(* IEC 61131-3 sources: RL_MAR/experiments/comparison/llm4plc/results/gpt-4o_20260507_114630/20260507_122226, 4 files *)

(* ---- generated_code_iteration_0.st ---- *)
plaintext
START_ST
FUNCTION_BLOCK AGVControlSystem
VAR_INPUT
    MaterialRequest : INT; (* New material handling request *)
END_VAR
VAR_OUTPUT
    AGV1_Ready : BOOL := TRUE; (* AGV 1 ready status *)
    AGV2_Ready : BOOL := TRUE; (* AGV 2 ready status *)
    AGV3_Ready : BOOL := TRUE; (* AGV 3 ready status *)
END_VAR
VAR
    state : INT := 0; (* Current state *)
    prevState : INT := 0; (* Previous state *)
    MaterialQueue : ARRAY[1..10] OF INT; (* FIFO queue for material requests *)
    queueHead : INT := 1; (* Points to the first element in the queue *)
    queueTail : INT := 0; (* Points to the last element in the queue *)
    AGVPosition : ARRAY[1..3] OF INT := [0, 0, 0]; (* Real-time AGV positions *)
    AGVStatus : ARRAY[1..3] OF BOOL := [TRUE, TRUE, TRUE]; (* Operational status of AGVs *)
    currentTask : ARRAY[1..3] OF INT := [0, 0, 0]; (* Task currently assigned to each AGV *)
    errorFlag : BOOL := FALSE; (* Error detection flag *)
    i : INT; (* Loop counter *)
END_VAR

(* Function to add a new material request to the queue *)
FUNCTION AddToQueue : BOOL
VAR_INPUT
    MaterialRequest : INT; (* Material request to be added *)
END_VAR
VAR
    success : BOOL := FALSE; (* Indicates if the operation was successful *)
END_VAR
IF queueTail < 10 THEN
    queueTail := queueTail + 1;
    MaterialQueue[queueTail] := MaterialRequest;
    success := TRUE;
ELSE
    success := FALSE; (* Queue overflow detected *)
END_IF
RETURN success;
END_FUNCTION

(* Function to assign tasks to AGVs based on priority and readiness *)
FUNCTION AssignTask : BOOL
VAR
    success : BOOL := FALSE; (* Indicates if the operation was successful *)
END_VAR
FOR i := 1 TO 3 DO
    IF AGVStatus[i] = TRUE AND queueHead <= queueTail THEN
        currentTask[i] := MaterialQueue[queueHead];
        AGVStatus[i] := FALSE; (* AGV is now working *)
        queueHead := queueHead + 1;
        success := TRUE;
        EXIT; (* Assign task to the highest priority AGV and exit *)
    END_IF
END_FOR
RETURN success;
END_FUNCTION

(* Function to update AGV position based on task progress *)
FUNCTION UpdateAGVPosition : BOOL
VAR_INPUT
    AGVIndex : INT; (* Index of the AGV to update *)
END_VAR
VAR
    success : BOOL := FALSE; (* Indicates if the operation was successful *)
END_VAR
IF AGVIndex >= 1 AND AGVIndex <= 3 THEN
    AGVPosition[AGVIndex] := AGVPosition[AGVIndex] + 1; (* Simulate position update *)
    IF AGVPosition[AGVIndex] < 0 THEN
        errorFlag := TRUE; (* Invalid position detected *)
        success := FALSE;
    ELSE
        success := TRUE;
    END_IF
END_IF
RETURN success;
END_FUNCTION

(* Function to reset AGV status after task completion *)
FUNCTION ResetAGVStatus : BOOL
VAR_INPUT
    AGVIndex : INT; (* Index of the AGV to reset *)
END_VAR
VAR
    success : BOOL := FALSE; (* Indicates if the operation was successful *)
END_VAR
IF AGVIndex >= 1 AND AGVIndex <= 3 THEN
    AGVStatus[AGVIndex] := TRUE; (* Reset AGV status to ready *)
    currentTask[AGVIndex] := 0; (* Clear the current task *)
    AGVPosition[AGVIndex] := 0; (* Reset position *)
    success := TRUE;
END_IF
RETURN success;
END_FUNCTION

(* Function to handle errors *)
FUNCTION HandleError : BOOL
VAR
    success : BOOL := FALSE; (* Indicates if the operation was successful *)
END_VAR
IF queueTail > 10 THEN
    queueTail := 10; (* Correct queue overflow *)
    errorFlag := TRUE;
    success := TRUE;
ELSIF errorFlag THEN
    errorFlag := FALSE; (* Clear error flag *)
    success := TRUE;
END_IF
RETURN success;
END_FUNCTION

(* Main logic for state transitions *)
CASE state OF
    0: (* IDLE *)
        IF MaterialRequest > 0 AND queueTail < 10 THEN
            prevState := state;
            state := 1; (* Transition to ADD_REQUEST_TO_QUEUE *)
        END_IF;
    1: (* ADD_REQUEST_TO_QUEUE *)
        IF AddToQueue(MaterialRequest) THEN
            prevState := state;
            state := 2; (* Transition to ASSIGN_TASK_TO_AGV *)
        ELSE
            prevState := state;
            state := 5; (* Transition to ERROR_HANDLING *)
        END_IF;
    2: (* ASSIGN_TASK_TO_AGV *)
        IF AssignTask() THEN
            prevState := state;
            state := 3; (* Transition to AGV_WORKING *)
        END_IF;
    3: (* AGV_WORKING *)
        FOR i := 1 TO 3 DO
            IF NOT AGVStatus[i] THEN
                IF UpdateAGVPosition(i) THEN
                    (* Check if task is completed *)
                    IF AGVPosition[i] >= 10 THEN
                        prevState := state;
                        state := 4; (* Transition to RESET_AGV_STATUS *)
                    END_IF;
                ELSE
                    prevState := state;
                    state := 5; (* Transition to ERROR_HANDLING *)
                END_IF;
            END_IF;
        END_FOR;
    4: (* RESET_AGV_STATUS *)
        FOR i := 1 TO 3 DO
            IF NOT AGVStatus[i] THEN
                IF ResetAGVStatus(i) THEN
                    prevState := state;
                    state := 0; (* Transition to IDLE *)
                END_IF;
            END_IF;
        END_FOR;
    5: (* ERROR_HANDLING *)
        IF HandleError() THEN
            prevState := state;
            state := 0; (* Transition to IDLE *)
        END_IF;
END_CASE;
END_FUNCTION_BLOCK
END_ST

(* ---- generated_code_iteration_1.st ---- *)
START_REASON
The feedback indicates that the `AddToQueue` function declaration is incorrect. Specifically, the function's output variable is improperly defined as `AddToQueue: BOOL;`. In Structured Text (ST), functions must use `VAR_OUTPUT` to declare output variables, not directly in the function header. This syntax error caused the CODESYS compiler validation to fail.

To resolve this issue, I will modify the function declaration to properly define the output variable using `VAR_OUTPUT`. Additionally, I will review the code for similar issues in other functions and ensure compliance with ST syntax standards.
END_REASON

START_ST
FUNCTION_BLOCK AGVControlSystem
VAR_INPUT
    MaterialRequest : INT; (* New material handling request *)
END_VAR
VAR_OUTPUT
    AGV1_Ready : BOOL := TRUE; (* AGV 1 ready status *)
    AGV2_Ready : BOOL := TRUE; (* AGV 2 ready status *)
    AGV3_Ready : BOOL := TRUE; (* AGV 3 ready status *)
END_VAR
VAR
    state : INT := 0; (* Current state *)
    prevState : INT := 0; (* Previous state *)
    MaterialQueue : ARRAY[1..10] OF INT; (* FIFO queue for material requests *)
    queueHead : INT := 1; (* Points to the first element in the queue *)
    queueTail : INT := 0; (* Points to the last element in the queue *)
    AGVPosition : ARRAY[1..3] OF INT := [0, 0, 0]; (* Real-time AGV positions *)
    AGVStatus : ARRAY[1..3] OF BOOL := [TRUE, TRUE, TRUE]; (* Operational status of AGVs *)
    currentTask : ARRAY[1..3] OF INT := [0, 0, 0]; (* Task currently assigned to each AGV *)
    errorFlag : BOOL := FALSE; (* Error detection flag *)
    i : INT; (* Loop counter *)
END_VAR

(* Function to add a new material request to the queue *)
FUNCTION AddToQueue : BOOL
VAR_INPUT
    MaterialRequest : INT; (* Material request to be added *)
END_VAR
VAR_OUTPUT
    success : BOOL; (* Indicates if the operation was successful *)
END_VAR
VAR
    tempSuccess : BOOL := FALSE; (* Temporary success flag *)
END_VAR
IF queueTail < 10 THEN
    queueTail := queueTail + 1;
    MaterialQueue[queueTail] := MaterialRequest;
    tempSuccess := TRUE;
ELSE
    tempSuccess := FALSE; (* Queue overflow detected *)
END_IF
success := tempSuccess;
RETURN success;
END_FUNCTION

(* Function to assign tasks to AGVs based on priority and readiness *)
FUNCTION AssignTask : BOOL
VAR_OUTPUT
    success : BOOL; (* Indicates if the operation was successful *)
END_VAR
VAR
    tempSuccess : BOOL := FALSE; (* Temporary success flag *)
END_VAR
FOR i := 1 TO 3 DO
    IF AGVStatus[i] = TRUE AND queueHead <= queueTail THEN
        currentTask[i] := MaterialQueue[queueHead];
        AGVStatus[i] := FALSE; (* AGV is now working *)
        queueHead := queueHead + 1;
        tempSuccess := TRUE;
        EXIT; (* Assign task to the highest priority AGV and exit *)
    END_IF
END_FOR
success := tempSuccess;
RETURN success;
END_FUNCTION

(* Function to update AGV position based on task progress *)
FUNCTION UpdateAGVPosition : BOOL
VAR_INPUT
    AGVIndex : INT; (* Index of the AGV to update *)
END_VAR
VAR_OUTPUT
    success : BOOL; (* Indicates if the operation was successful *)
END_VAR
VAR
    tempSuccess : BOOL := FALSE; (* Temporary success flag *)
END_VAR
IF AGVIndex >= 1 AND AGVIndex <= 3 THEN
    AGVPosition[AGVIndex] := AGVPosition[AGVIndex] + 1; (* Simulate position update *)
    IF AGVPosition[AGVIndex] < 0 THEN
        errorFlag := TRUE; (* Invalid position detected *)
        tempSuccess := FALSE;
    ELSE
        tempSuccess := TRUE;
    END_IF
END_IF
success := tempSuccess;
RETURN success;
END_FUNCTION

(* Function to reset AGV status after task completion *)
FUNCTION ResetAGVStatus : BOOL
VAR_INPUT
    AGVIndex : INT; (* Index of the AGV to reset *)
END_VAR
VAR_OUTPUT
    success : BOOL; (* Indicates if the operation was successful *)
END_VAR
VAR
    tempSuccess : BOOL := FALSE; (* Temporary success flag *)
END_VAR
IF AGVIndex >= 1 AND AGVIndex <= 3 THEN
    AGVStatus[AGVIndex] := TRUE; (* Reset AGV status to ready *)
    currentTask[AGVIndex] := 0; (* Clear the current task *)
    AGVPosition[AGVIndex] := 0; (* Reset position *)
    tempSuccess := TRUE;
END_IF
success := tempSuccess;
RETURN success;
END_FUNCTION

(* Function to handle errors *)
FUNCTION HandleError : BOOL
VAR_OUTPUT
    success : BOOL; (* Indicates if the operation was successful *)
END_VAR
VAR
    tempSuccess : BOOL := FALSE; (* Temporary success flag *)
END_VAR
IF queueTail > 10 THEN
    queueTail := 10; (* Correct queue overflow *)
    errorFlag := TRUE;
    tempSuccess := TRUE;
ELSIF errorFlag THEN
    errorFlag := FALSE; (* Clear error flag *)
    tempSuccess := TRUE;
END_IF
success := tempSuccess;
RETURN success;
END_FUNCTION

(* Main logic for state transitions *)
CASE state OF
    0: (* IDLE *)
        IF MaterialRequest > 0 AND queueTail < 10 THEN
            prevState := state;
            state := 1; (* Transition to ADD_REQUEST_TO_QUEUE *)
        END_IF;
    1: (* ADD_REQUEST_TO_QUEUE *)
        IF AddToQueue(MaterialRequest) THEN
            prevState := state;
            state := 2; (* Transition to ASSIGN_TASK_TO_AGV *)
        ELSE
            prevState := state;
            state := 5; (* Transition to ERROR_HANDLING *)
        END_IF;
    2: (* ASSIGN_TASK_TO_AGV *)
        IF AssignTask() THEN
            prevState := state;
            state := 3; (* Transition to AGV_WORKING *)
        END_IF;
    3: (* AGV_WORKING *)
        FOR i := 1 TO 3 DO
            IF NOT AGVStatus[i] THEN
                IF UpdateAGVPosition(i) THEN
                    (* Check if task is completed *)
                    IF AGVPosition[i] >= 10 THEN
                        prevState := state;
                        state := 4; (* Transition to RESET_AGV_STATUS *)
                    END_IF;
                ELSE
                    prevState := state;
                    state := 5; (* Transition to ERROR_HANDLING *)
                END_IF;
            END_IF;
        END_FOR;
    4: (* RESET_AGV_STATUS *)
        FOR i := 1 TO 3 DO
            IF NOT AGVStatus[i] THEN
                IF ResetAGVStatus(i) THEN
                    prevState := state;
                    state := 0; (* Transition to IDLE *)
                END_IF;
            END_IF;
        END_FOR;
    5: (* ERROR_HANDLING *)
        IF HandleError() THEN
            prevState := state;
            state := 0; (* Transition to IDLE *)
        END_IF;
END_CASE;
END_FUNCTION_BLOCK
END_ST

(* ---- generated_code_iteration_2.st ---- *)
START_REASON
The feedback indicates that the `AddToQueue` function declaration is incorrect due to the improper definition of the output variable as `AddToQueue: BOOL;`. In Structured Text (ST), functions must use `VAR_OUTPUT` to declare output variables, not directly in the function header. This syntax error caused the CODESYS compiler validation to fail.

To resolve this issue, I will modify the `AddToQueue` function declaration to properly define the output variable using `VAR_OUTPUT`. Additionally, I will ensure that all functions follow the correct ST syntax standards and review the code for similar issues in other functions. This will ensure compliance with the CODESYS compiler requirements.
END_REASON

START_ST
FUNCTION_BLOCK AGVControlSystem
VAR_INPUT
    MaterialRequest : INT; (* New material handling request *)
END_VAR
VAR_OUTPUT
    AGV1_Ready : BOOL := TRUE; (* AGV 1 ready status *)
    AGV2_Ready : BOOL := TRUE; (* AGV 2 ready status *)
    AGV3_Ready : BOOL := TRUE; (* AGV 3 ready status *)
END_VAR
VAR
    state : INT := 0; (* Current state *)
    prevState : INT := 0; (* Previous state *)
    MaterialQueue : ARRAY[1..10] OF INT; (* FIFO queue for material requests *)
    queueHead : INT := 1; (* Points to the first element in the queue *)
    queueTail : INT := 0; (* Points to the last element in the queue *)
    AGVPosition : ARRAY[1..3] OF INT := [0, 0, 0]; (* Real-time AGV positions *)
    AGVStatus : ARRAY[1..3] OF BOOL := [TRUE, TRUE, TRUE]; (* Operational status of AGVs *)
    currentTask : ARRAY[1..3] OF INT := [0, 0, 0]; (* Task currently assigned to each AGV *)
    errorFlag : BOOL := FALSE; (* Error detection flag *)
    i : INT; (* Loop counter *)
END_VAR

(* Function to add a new material request to the queue *)
FUNCTION AddToQueue
VAR_INPUT
    MaterialRequest : INT; (* Material request to be added *)
END_VAR
VAR_OUTPUT
    success : BOOL; (* Indicates if the operation was successful *)
END_VAR
VAR
    tempSuccess : BOOL := FALSE; (* Temporary success flag *)
END_VAR
IF queueTail < 10 THEN
    queueTail := queueTail + 1;
    MaterialQueue[queueTail] := MaterialRequest;
    tempSuccess := TRUE;
ELSE
    tempSuccess := FALSE; (* Queue overflow detected *)
END_IF
success := tempSuccess;
RETURN success;
END_FUNCTION

(* Function to assign tasks to AGVs based on priority and readiness *)
FUNCTION AssignTask
VAR_OUTPUT
    success : BOOL; (* Indicates if the operation was successful *)
END_VAR
VAR
    tempSuccess : BOOL := FALSE; (* Temporary success flag *)
END_VAR
FOR i := 1 TO 3 DO
    IF AGVStatus[i] = TRUE AND queueHead <= queueTail THEN
        currentTask[i] := MaterialQueue[queueHead];
        AGVStatus[i] := FALSE; (* AGV is now working *)
        queueHead := queueHead + 1;
        tempSuccess := TRUE;
        EXIT; (* Assign task to the highest priority AGV and exit *)
    END_IF
END_FOR
success := tempSuccess;
RETURN success;
END_FUNCTION

(* Function to update AGV position based on task progress *)
FUNCTION UpdateAGVPosition
VAR_INPUT
    AGVIndex : INT; (* Index of the AGV to update *)
END_VAR
VAR_OUTPUT
    success : BOOL; (* Indicates if the operation was successful *)
END_VAR
VAR
    tempSuccess : BOOL := FALSE; (* Temporary success flag *)
END_VAR
IF AGVIndex >= 1 AND AGVIndex <= 3 THEN
    AGVPosition[AGVIndex] := AGVPosition[AGVIndex] + 1; (* Simulate position update *)
    IF AGVPosition[AGVIndex] < 0 THEN
        errorFlag := TRUE; (* Invalid position detected *)
        tempSuccess := FALSE;
    ELSE
        tempSuccess := TRUE;
    END_IF
END_IF
success := tempSuccess;
RETURN success;
END_FUNCTION

(* Function to reset AGV status after task completion *)
FUNCTION ResetAGVStatus
VAR_INPUT
    AGVIndex : INT; (* Index of the AGV to reset *)
END_VAR
VAR_OUTPUT
    success : BOOL; (* Indicates if the operation was successful *)
END_VAR
VAR
    tempSuccess : BOOL := FALSE; (* Temporary success flag *)
END_VAR
IF AGVIndex >= 1 AND AGVIndex <= 3 THEN
    AGVStatus[AGVIndex] := TRUE; (* Reset AGV status to ready *)
    currentTask[AGVIndex] := 0; (* Clear the current task *)
    AGVPosition[AGVIndex] := 0; (* Reset position *)
    tempSuccess := TRUE;
END_IF
success := tempSuccess;
RETURN success;
END_FUNCTION

(* Function to handle errors *)
FUNCTION HandleError
VAR_OUTPUT
    success : BOOL; (* Indicates if the operation was successful *)
END_VAR
VAR
    tempSuccess : BOOL := FALSE; (* Temporary success flag *)
END_VAR
IF queueTail > 10 THEN
    queueTail := 10; (* Correct queue overflow *)
    errorFlag := TRUE;
    tempSuccess := TRUE;
ELSIF errorFlag THEN
    errorFlag := FALSE; (* Clear error flag *)
    tempSuccess := TRUE;
END_IF
success := tempSuccess;
RETURN success;
END_FUNCTION

(* Main logic for state transitions *)
CASE state OF
    0: (* IDLE *)
        IF MaterialRequest > 0 AND queueTail < 10 THEN
            prevState := state;
            state := 1; (* Transition to ADD_REQUEST_TO_QUEUE *)
        END_IF;
    1: (* ADD_REQUEST_TO_QUEUE *)
        IF AddToQueue(MaterialRequest) THEN
            prevState := state;
            state := 2; (* Transition to ASSIGN_TASK_TO_AGV *)
        ELSE
            prevState := state;
            state := 5; (* Transition to ERROR_HANDLING *)
        END_IF;
    2: (* ASSIGN_TASK_TO_AGV *)
        IF AssignTask() THEN
            prevState := state;
            state := 3; (* Transition to AGV_WORKING *)
        END_IF;
    3: (* AGV_WORKING *)
        FOR i := 1 TO 3 DO
            IF NOT AGVStatus[i] THEN
                IF UpdateAGVPosition(i) THEN
                    (* Check if task is completed *)
                    IF AGVPosition[i] >= 10 THEN
                        prevState := state;
                        state := 4; (* Transition to RESET_AGV_STATUS *)
                    END_IF;
                ELSE
                    prevState := state;
                    state := 5; (* Transition to ERROR_HANDLING *)
                END_IF;
            END_IF;
        END_FOR;
    4: (* RESET_AGV_STATUS *)
        FOR i := 1 TO 3 DO
            IF NOT AGVStatus[i] THEN
                IF ResetAGVStatus(i) THEN
                    prevState := state;
                    state := 0; (* Transition to IDLE *)
                END_IF;
            END_IF;
        END_FOR;
    5: (* ERROR_HANDLING *)
        IF HandleError() THEN
            prevState := state;
            state := 0; (* Transition to IDLE *)
        END_IF;
END_CASE;
END_FUNCTION_BLOCK
END_ST

(* ---- generated_code_iteration_3.st ---- *)
START_REASON
The feedback indicates that the `AddToQueue` function declaration incorrectly defines the output variable directly in the function header (`AddToQueue: BOOL;`). In Structured Text (ST), output variables must be declared using `VAR_OUTPUT` instead of directly in the function header. This syntax error caused the CODESYS compiler validation to fail.

To resolve this issue, I will ensure that all functions, including `AddToQueue`, follow the correct ST syntax standards. Specifically, I will modify the `AddToQueue` function to properly define the output variable using `VAR_OUTPUT`. Additionally, I will review the code for similar issues in other functions and ensure compliance with the CODESYS compiler requirements.
END_REASON

START_ST
FUNCTION_BLOCK AGVControlSystem
VAR_INPUT
    MaterialRequest : INT; (* New material handling request *)
END_VAR
VAR_OUTPUT
    AGV1_Ready : BOOL := TRUE; (* AGV 1 ready status *)
    AGV2_Ready : BOOL := TRUE; (* AGV 2 ready status *)
    AGV3_Ready : BOOL := TRUE; (* AGV 3 ready status *)
END_VAR
VAR
    state : INT := 0; (* Current state *)
    prevState : INT := 0; (* Previous state *)
    MaterialQueue : ARRAY[1..10] OF INT; (* FIFO queue for material requests *)
    queueHead : INT := 1; (* Points to the first element in the queue *)
    queueTail : INT := 0; (* Points to the last element in the queue *)
    AGVPosition : ARRAY[1..3] OF INT := [0, 0, 0]; (* Real-time AGV positions *)
    AGVStatus : ARRAY[1..3] OF BOOL := [TRUE, TRUE, TRUE]; (* Operational status of AGVs *)
    currentTask : ARRAY[1..3] OF INT := [0, 0, 0]; (* Task currently assigned to each AGV *)
    errorFlag : BOOL := FALSE; (* Error detection flag *)
    i : INT; (* Loop counter *)
END_VAR

(* Function to add a new material request to the queue *)
FUNCTION AddToQueue : BOOL
VAR_INPUT
    MaterialRequest : INT; (* Material request to be added *)
END_VAR
VAR_OUTPUT
    success : BOOL; (* Indicates if the operation was successful *)
END_VAR
VAR
    tempSuccess : BOOL := FALSE; (* Temporary success flag *)
END_VAR
IF queueTail < 10 THEN
    queueTail := queueTail + 1;
    MaterialQueue[queueTail] := MaterialRequest;
    tempSuccess := TRUE;
ELSE
    tempSuccess := FALSE; (* Queue overflow detected *)
END_IF
success := tempSuccess;
RETURN success;
END_FUNCTION

(* Function to assign tasks to AGVs based on priority and readiness *)
FUNCTION AssignTask : BOOL
VAR_OUTPUT
    success : BOOL; (* Indicates if the operation was successful *)
END_VAR
VAR
    tempSuccess : BOOL := FALSE; (* Temporary success flag *)
END_VAR
FOR i := 1 TO 3 DO
    IF AGVStatus[i] = TRUE AND queueHead <= queueTail THEN
        currentTask[i] := MaterialQueue[queueHead];
        AGVStatus[i] := FALSE; (* AGV is now working *)
        queueHead := queueHead + 1;
        tempSuccess := TRUE;
        EXIT; (* Assign task to the highest priority AGV and exit *)
    END_IF
END_FOR
success := tempSuccess;
RETURN success;
END_FUNCTION

(* Function to update AGV position based on task progress *)
FUNCTION UpdateAGVPosition : BOOL
VAR_INPUT
    AGVIndex : INT; (* Index of the AGV to update *)
END_VAR
VAR_OUTPUT
    success : BOOL; (* Indicates if the operation was successful *)
END_VAR
VAR
    tempSuccess : BOOL := FALSE; (* Temporary success flag *)
END_VAR
IF AGVIndex >= 1 AND AGVIndex <= 3 THEN
    AGVPosition[AGVIndex] := AGVPosition[AGVIndex] + 1; (* Simulate position update *)
    IF AGVPosition[AGVIndex] < 0 THEN
        errorFlag := TRUE; (* Invalid position detected *)
        tempSuccess := FALSE;
    ELSE
        tempSuccess := TRUE;
    END_IF
END_IF
success := tempSuccess;
RETURN success;
END_FUNCTION

(* Function to reset AGV status after task completion *)
FUNCTION ResetAGVStatus : BOOL
VAR_INPUT
    AGVIndex : INT; (* Index of the AGV to reset *)
END_VAR
VAR_OUTPUT
    success : BOOL; (* Indicates if the operation was successful *)
END_VAR
VAR
    tempSuccess : BOOL := FALSE; (* Temporary success flag *)
END_VAR
IF AGVIndex >= 1 AND AGVIndex <= 3 THEN
    AGVStatus[AGVIndex] := TRUE; (* Reset AGV status to ready *)
    currentTask[AGVIndex] := 0; (* Clear the current task *)
    AGVPosition[AGVIndex] := 0; (* Reset position *)
    tempSuccess := TRUE;
END_IF
success := tempSuccess;
RETURN success;
END_FUNCTION

(* Function to handle errors *)
FUNCTION HandleError : BOOL
VAR_OUTPUT
    success : BOOL; (* Indicates if the operation was successful *)
END_VAR
VAR
    tempSuccess : BOOL := FALSE; (* Temporary success flag *)
END_VAR
IF queueTail > 10 THEN
    queueTail := 10; (* Correct queue overflow *)
    errorFlag := TRUE;
    tempSuccess := TRUE;
ELSIF errorFlag THEN
    errorFlag := FALSE; (* Clear error flag *)
    tempSuccess := TRUE;
END_IF
success := tempSuccess;
RETURN success;
END_FUNCTION

(* Main logic for state transitions *)
CASE state OF
    0: (* IDLE *)
        IF MaterialRequest > 0 AND queueTail < 10 THEN
            prevState := state;
            state := 1; (* Transition to ADD_REQUEST_TO_QUEUE *)
        END_IF;
    1: (* ADD_REQUEST_TO_QUEUE *)
        IF AddToQueue(MaterialRequest) THEN
            prevState := state;
            state := 2; (* Transition to ASSIGN_TASK_TO_AGV *)
        ELSE
            prevState := state;
            state := 5; (* Transition to ERROR_HANDLING *)
        END_IF;
    2: (* ASSIGN_TASK_TO_AGV *)
        IF AssignTask() THEN
            prevState := state;
            state := 3; (* Transition to AGV_WORKING *)
        END_IF;
    3: (* AGV_WORKING *)
        FOR i := 1 TO 3 DO
            IF NOT AGVStatus[i] THEN
                IF UpdateAGVPosition(i) THEN
                    (* Check if task is completed *)
                    IF AGVPosition[i] >= 10 THEN
                        prevState := state;
                        state := 4; (* Transition to RESET_AGV_STATUS *)
                    END_IF;
                ELSE
                    prevState := state;
                    state := 5; (* Transition to ERROR_HANDLING *)
                END_IF;
            END_IF;
        END_FOR;
    4: (* RESET_AGV_STATUS *)
        FOR i := 1 TO 3 DO
            IF NOT AGVStatus[i] THEN
                IF ResetAGVStatus(i) THEN
                    prevState := state;
                    state := 0; (* Transition to IDLE *)
                END_IF;
            END_IF;
        END_FOR;
    5: (* ERROR_HANDLING *)
        IF HandleError() THEN
            prevState := state;
            state := 0; (* Transition to IDLE *)
        END_IF;
END_CASE;
END_FUNCTION_BLOCK
END_ST
